Staubli VAL3: getIO.pgx

public program getIO(string& x_sIO)
begin
  x_sIO=sIOName
end
